Yaskawa INFORM job: TWIN_FRONT_SEARCH_90ST-2_5340.JBI

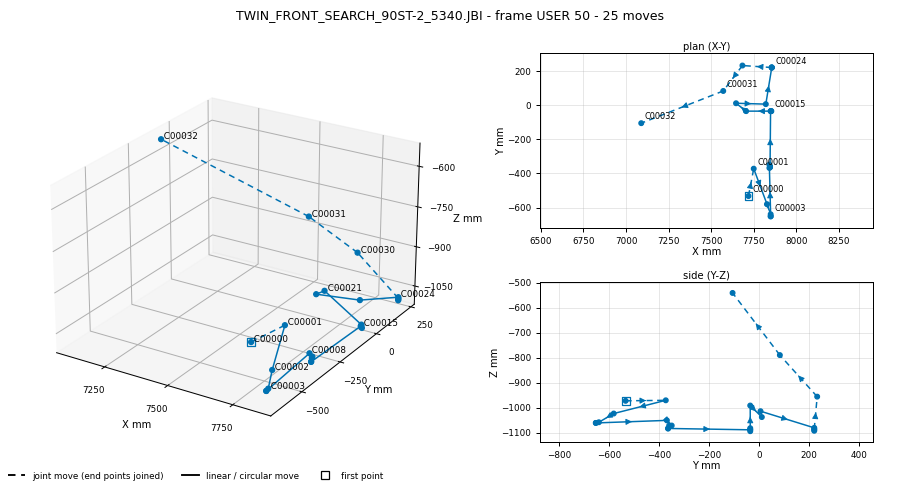
[picture p0: tool path of TWIN_FRONT_SEARCH_90ST-2_5340.JBI in frame USER 50, 25 of 25 moves have a stored position in this frame; points joined in program order, loops and branches not executed]
/JOB
//NAME TWIN_FRONT_SEARCH_90ST-2_5340
///FOLDERNAME 02-SKRZYNIE_JOBS
//POS
///NPOS 33,33,0,5,0,0
///USER 50
///TOOL 0
///POSTYPE USER
///RECTAN
///RCONF 1,0,0,0,0,0,0,0,0,0,0,0,0,0,0,0,0,0,0,0,0,0,0,0
C00000=7719.055,-532.713,-972.768,-40.3407,48.0630,66.6722
///RCONF 0,0,0,0,0,0,0,0,0,0,0,0,0,0,0,0,0,0,0,0,0,0,0,0
C00001=7749.941,-372.029,-970.713,-33.2752,28.4585,82.6051
C00002=7827.863,-580.311,-1023.644,-35.7540,43.0939,104.6870
C00003=7849.471,-639.809,-1058.524,-35.7541,43.0927,104.6878
C00004=7849.503,-639.771,-1072.165,-35.7563,43.0913,104.6874
C00005=7849.523,-651.960,-1061.282,-35.7586,43.0891,104.6854
C00006=7861.907,-651.998,-1061.296,-35.7586,43.0886,104.6813
C00007=7849.523,-651.960,-1061.282,-35.7586,43.0891,104.6854
C00008=7841.995,-367.647,-1051.045,-35.7572,43.0898,104.6866
C00009=7841.992,-348.302,-1071.676,-35.7565,43.0913,104.6877
C00010=7845.832,-358.396,-1071.678,-35.7555,43.0924,104.6885
C00011=7845.819,-358.421,-1091.925,-35.7551,43.0900,104.6820
C00012=7845.831,-362.847,-1083.353,-35.7564,43.0898,104.6825
C00013=7863.182,-362.835,-1083.347,-35.7564,43.0895,104.6832
C00014=7845.831,-362.847,-1083.353,-35.7564,43.0898,104.6825
///RCONF 1,0,0,0,0,0,0,0,0,0,0,0,0,0,0,0,0,0,0,0,0,0,0,0
C00015=7848.879,-34.086,-1088.772,-31.8323,42.1270,99.9912
C00016=7851.273,-34.077,-1087.501,-31.8321,42.1263,99.9914
C00017=7851.280,-34.079,-1097.582,-31.8328,42.1254,99.9896
C00018=7853.474,-34.063,-1094.331,-31.8298,42.1250,99.9939
C00019=7866.095,-34.062,-1094.352,-31.8295,42.1238,99.9919
C00020=7851.277,-34.079,-1082.326,-31.8318,42.1273,99.9920
///RCONF 0,0,0,0,0,0,0,0,0,0,0,0,0,0,0,0,0,0,0,0,0,0,0,0
C00021=7705.283,-34.120,-991.640,-31.8316,42.1293,99.9928
C00022=7646.131,12.247,-1037.802,-5.9165,-10.8227,-7.1237
///RCONF 1,0,0,0,0,0,0,0,0,0,0,0,0,0,0,0,0,0,0,0,0,0,0,0
C00023=7820.935,7.066,-1014.348,37.0724,25.7387,-108.9100
C00024=7855.836,222.083,-1080.856,23.4711,44.5719,-116.2729
C00025=7855.862,222.072,-1088.838,23.4734,44.5725,-116.2722
C00026=7855.849,222.057,-1096.938,23.4735,44.5708,-116.2706
C00027=7855.835,222.050,-1092.624,23.4716,44.5706,-116.2731
C00028=7866.915,222.052,-1092.630,23.4699,44.5708,-116.2753
C00029=7855.856,222.058,-1085.089,23.4748,44.5706,-116.2687
C00030=7683.667,233.765,-956.083,23.4688,44.5707,-116.2734
C00031=7570.947,84.363,-789.769,8.3295,54.7414,-178.0447
C00032=7089.401,-104.773,-541.114,-34.6747,-14.1850,36.1511
///RCONF 0,0,0,0,0,0,0,0,0,0,0,0,0,0,0,0,0,0,0,0,0,0,0,0
BC00000=6307.477
BC00001=6307.477
BC00002=6515.049
BC00003=6515.049
BC00004=6515.049
BC00005=6515.049
BC00006=6515.049
BC00007=6515.049
BC00008=6515.049
BC00009=6515.049
BC00010=6515.049
BC00011=6515.049
BC00012=6515.049
BC00013=6515.049
BC00014=6515.049
BC00015=6515.049
BC00016=6515.049
BC00017=6515.049
BC00018=6515.049
BC00019=6515.049
BC00020=6515.049
BC00021=6515.049
BC00022=6515.049
BC00023=6515.049
BC00024=6515.049
BC00025=6515.049
BC00026=6515.049
BC00027=6515.049
BC00028=6515.049
BC00029=6515.049
BC00030=6428.036
BC00031=6132.885
BC00032=5388.459
///POSTYPE BASE
P00006=-2.449,0.031,8.825,0.0000,0.0000,0.0000
P00501=-2.026,0.009,3.534,0.0000,0.0000,0.0000
///RCONF 1,0,0,0,0,0,0,0,0,0,0,0,0,0,0,0,0,0,0,0,0,0,0,0
P00502=-2.023,0.001,1.732,0.0000,0.0000,0.0000
P00503=0.138,-0.044,1.539,0.0000,0.0000,0.0000
P00504=-0.309,-0.010,1.636,0.0000,0.0000,0.0000
//INST
///DATE 2024/10/29 09:28
///ATTR SC,RW,RJ
////FRAME USER 50
///GROUP1 RB1,BS1
NOP
MOVJ C00000 BC00000 VJ=80.00
MOVJ C00001 BC00001 VJ=40.00
'::::::::::::::::::::::::::::::::
'W56 P
'::::::::::::::::::::::::::::::::
MOVL C00002 BC00002 V=500.0
SFTOF
MOVL C00003 BC00003 V=166.7 PL=0
REFP 3 C00004 BC00004
CALL JOB:SEARCH-R1
SET P0501 P0006
SFTON P0501
MOVL C00005 BC00005 V=166.7 PL=0
REFP 3 C00006 BC00006
CALL JOB:SEARCH-R1
SET P0501 P0006
SFTON P0501
MOVL C00007 BC00007 V=250.0 PL=0
SFTOF
MOVL C00008 BC00008 V=333.3
'::::::::::::::::::::::::::::::::
'W56 L
'::::::::::::::::::::::::::::::::
MOVL C00009 BC00009 V=333.3
MOVL C00010 BC00010 V=166.7 PL=0
REFP 3 C00011 BC00011
CALL JOB:SEARCH-R1
SET P0502 P0006
SFTON P0502
MOVL C00012 BC00012 V=166.7 PL=0
REFP 3 C00013 BC00013
CALL JOB:SEARCH-R1
SET P0502 P0006
SFTON P0502
MOVL C00014 BC00014 V=250.0 PL=0
SFTOF
'::::::::::::::::::::::::::::::::
'W57 P
'::::::::::::::::::::::::::::::::
MOVL C00015 BC00015 V=500.0
MOVL C00016 BC00016 V=100.0 PL=0
REFP 3 C00017 BC00017
CALL JOB:SEARCH-R1
SET P0503 P0006
SFTON P0503
MOVL C00018 BC00018 V=166.7 PL=0
REFP 3 C00019 BC00019
CALL JOB:SEARCH-R1
SET P0503 P0006
SFTON P0503
MOVL C00020 BC00020 V=250.0 PL=0
SFTOF
'::::::::::::::::::::::::::::::::
'W57 L
'::::::::::::::::::::::::::::::::
MOVL C00021 BC00021 V=333.3
MOVL C00022 BC00022 V=333.3
MOVL C00023 BC00023 V=333.3
MOVL C00024 BC00024 V=500.0
MOVL C00025 BC00025 V=166.7 PL=0
REFP 3 C00026 BC00026
CALL JOB:SEARCH-R1
SET P0504 P0006
SFTON P0504
MOVL C00027 BC00027 V=166.7 PL=0
REFP 3 C00028 BC00028
CALL JOB:SEARCH-R1
SET P0504 P0006
SFTON P0504
MOVL C00029 BC00029 V=250.0 PL=0
SFTOF
MOVJ C00030 BC00030 VJ=50.00
MOVJ C00031 BC00031 VJ=50.00
MOVJ C00032 BC00032 VJ=80.00
END
